{attribute 'analysis' := '-33'}
PROGRAM INTERNAL PRG_EnumTests
VAR
{IF defined (UNIT_TEST)}
	fbF_ComputeEnumSizeTests : FB_F_ComputeEnumSizeTests;
{END_IF}
END_VAR

END_PROGRAM

(* stored: Version 1.1.0.1
   POU PRG_EnumTests: Id {ceba0ca6-59f4-431a-b804-f579676d862c}, SpecialFunc None *)
